INTERFACE I_Mover

METHOD CycleUpdate : BOOL
VAR_INPUT
END_VAR
END_METHOD

METHOD Init : BOOL
VAR_INPUT
	XtsMover:  I_XtsXlMover1;
	XtsProcessingUnit :  I_XtsProcessingUnit1;
END_VAR
END_METHOD

METHOD JoinNearestTrack : BOOL


VAR

END_VAR
END_METHOD

METHOD LeaveSystemAt : BOOL
VAR_INPUT
	ConnectionOut: REFERENCE TO MC_PlanarTrackConnectionOut;	
END_VAR
END_METHOD

METHOD MoveOnTrack : BOOL
VAR_INPUT
	track: REFERENCE TO MC_PlanarTrack;	
	targetPos: LREAL;
	gap : LREAL; 
	velo : LREAL; 
END_VAR
END_METHOD

PROPERTY MoverOTCID : OTCID
GET
END_GET
SET
END_SET
END_PROPERTY

PROPERTY MoverStopped : BOOL
GET
END_GET
SET
END_SET
END_PROPERTY

PROPERTY P_Dynamics : REFERENCE TO DynamicConstraint_PathXY;
GET
END_GET
END_PROPERTY

PROPERTY P_InSync : Bool
GET
END_GET
END_PROPERTY

PROPERTY P_PlanarFeedback : REFERENCE TO MC_PlanarFeedback
GET
END_GET
END_PROPERTY

PROPERTY P_PlanarMover :   REFERENCE TO  MC_PlanarMover
GET
END_GET
END_PROPERTY

PROPERTY P_TargetTrack : UDINT
GET
END_GET
SET
END_SET
END_PROPERTY

PROPERTY Rework : BOOL
GET
END_GET
SET
END_SET
END_PROPERTY

METHOD SyncToOtherMover : Bool
VAR_INPUT
	masterSyncPos : LREAL; // Position on the master track
	followerSyncPos : LREAL; // position on the follower track
	PlanarMoverToFollow: REFERENCE TO Tc3_Mc3PlanarMotion.MC_PlanarMover;
	masterTrack : REFERENCE TO Tc3_Mc3PlanarMotion.MC_PlanarTrack; 
	followerTrack : REFERENCE TO Tc3_Mc3PlanarMotion.MC_PlanarTrack; 
	velo : LREAL; 
END_VAR
END_METHOD

METHOD  UpdateXtsTrack
VAR_INPUT
END_VAR
VAR

END_VAR
END_METHOD

PROPERTY XlProcessingUnit : I_XtsProcessingUnit1
GET
END_GET
END_PROPERTY

PROPERTY XtsComFeed : REFERENCE TO  XtsCommandFeedback
GET
END_GET
END_PROPERTY

PROPERTY XtsXlMover :  I_XtsXlMover1
GET
END_GET
END_PROPERTY

END_INTERFACE

(* stored: Version 1.1.0.1
   Itf I_Mover: Id {b268cb59-d99c-43ca-ba0f-41461eab83e4}
   Method CycleUpdate: Id {48e7b414-8a52-4904-8a2c-941ff8cf97f0}
   Method Init: Id {70e27be2-2f8a-4a12-af9c-c87e7a1f6409}
   Method JoinNearestTrack: Id {1af77ee2-ffb0-46d3-b285-380f37f7d28e}
   Method LeaveSystemAt: Id {b24f1fa5-5146-4fc9-b97d-6c3d7849e67f}
   Method MoveOnTrack: Id {c4ca36ea-3628-4f8d-9779-76967292fe61}
   Property MoverOTCID: Id {48d62f0a-81b1-4685-945a-1fd17f9606ba}
   Get Get: Id {e1662943-3496-4c10-924b-632c7ff27b5f}
   Set Set: Id {36ee8c57-942c-41b5-9bcd-87fb52eeb16e}
   Property MoverStopped: Id {9803e80b-12ab-4e37-a4f8-315195184be1}
   Get Get: Id {35a05db8-9b6b-41a5-81d3-287cc15ec088}
   Set Set: Id {1f4968b4-7a34-4354-9095-a9931b065151}
   Property P_Dynamics: Id {a2d4066c-df4e-4534-b63b-1bcfe3693364}
   Get Get: Id {b36cac87-776c-416b-845f-0437976c5461}
   Property P_InSync: Id {44e12130-9d7b-42f1-8fbe-83c3e8bf9e21}
   Get Get: Id {c1e62b68-c344-428b-816f-4dc4e05c9105}
   Property P_PlanarFeedback: Id {9e77b007-b995-4d4e-847f-52481bc8b65f}
   Get Get: Id {e9ed8e49-d6ca-4f9e-8d3e-078d51cca372}
   Property P_PlanarMover: Id {fa6a8c9a-a607-48a6-a503-b7396c44d435}
   Get Get: Id {026c43a2-9a34-4289-9222-3635d4914500}
   Property P_TargetTrack: Id {efe12142-6a27-4117-844c-b25d6699356f}
   Get Get: Id {050e7b0f-6fb8-46ed-b024-1523fc1288a0}
   Set Set: Id {d595508e-dce0-4463-ba46-7e3d11bc7415}
   Property Rework: Id {0cbdc2c5-5567-4b77-b67c-5f6aa39ca7ad}
   Get Get: Id {b67ca10e-23ed-42ec-9173-14befebfdf86}
   Set Set: Id {84e8a0f5-3c75-4d33-9ae3-4c9b7c60c721}
   Method SyncToOtherMover: Id {53951dae-e642-4c0f-afd2-22812dd067a9}
   Method UpdateXtsTrack: Id {f15d0a33-41f6-42cf-a0d1-8e20b2064dca}
   Property XlProcessingUnit: Id {4fb3d0ec-89c3-4528-ba23-e01b215f5acc}
   Get Get: Id {6ac1a39c-60c2-4a86-96ab-c6cda818fea0}
   Property XtsComFeed: Id {9b70f023-8c1f-45c7-92b4-2da0d8c5dc09}
   Get Get: Id {bfdc277d-d5e2-4691-a07e-5ee73b6a008d}
   Property XtsXlMover: Id {bb8d0ca5-767e-4004-9c86-a2c6dc44ab36}
   Get Get: Id {6829a4d3-d4f9-4a18-8081-1eebf326643d} *)
